{attribute 'GeneratedUsingTerminal: EL3773-0000-0018'}
{attribute addProperty BoxType "EL3773-0000-0018"}
{attribute addProperty Id "U1_SamplesAT %I*U1_Samples_2D13B74B20"}
{attribute addProperty CRC "2456502413"}
{attribute addProperty Size "20"}
TYPE L1_Voltage_Samples_926B408D :
STRUCT
	{attribute addProperty Name "U1_Samples"}
	U1_Samples AT %I* : U1_Samples_2D13B74B;
END_STRUCT
END_TYPE

(* stored: Version 1.2.0.0, ProductVersion 3.1.4024.9
   DUT L1_Voltage_Samples_926B408D: Id {4c8b7171-301b-45ee-a978-b0b2f2f47306} *)
